// TIA Portal V16 export
// export: Created 2024-09-05T17:36:33.3878466Z, ExportSetting WithDefaults, DisplayName Totally Integrated Automation Portal, DisplayVersion V16 Update 6, DisplayName TIA Portal Version Control Interface, DisplayVersion V16 Update 2, DisplayName TIA Portal Openness, DisplayVersion V16 Update 6, DisplayName STEP 7 Professional, DisplayVersion V16 Update 6, DisplayName STEP 7 Safety, DisplayVersion V16, DisplayName WinCC Advanced, DisplayVersion V16 Update 6
VAR_GLOBAL   // PLC tag table "IO"
   iNokBoxPresent AT %I27.4 : Bool;
   iNokPartOpticalSensor AT %I27.6 : Bool;
END_VAR
VAR_GLOBAL CONSTANT   // user constants
   IOImageSize : Int := 20;
END_VAR
